FUNCTION F_ComputeBoolSize : UDINT
VAR_INPUT
    {attribute 'analysis' := '-33' }
    bValue : BOOL;
END_VAR


F_ComputeBoolSize := GCL_PB.cBoolSize;

END_FUNCTION

(* stored: Version 1.1.0.1
   POU F_ComputeBoolSize: Id {147bcd4c-9238-47d3-a897-e3b625829b50}, SpecialFunc None *)
